# EPICS autosave request: iocBoot/ioc13bmd/auto_positions.req
file "CARS_80_motor_positions.req", P=$(P)
